{attribute 'GeneratedUsingTerminal: EL2032--0000'}
{attribute addProperty BoxType "EL2032--0000"}
{attribute addProperty Id "DiagAT %I*BOOL1"}
{attribute addProperty CRC "2804620823"}
{attribute addProperty Size "1"}
TYPE Diag_A72B1E17 EXTENDS InputBase_8311D824 :
STRUCT
	{attribute addProperty Name "Diag"}
	Diag AT %I* : BOOL;
END_STRUCT
END_TYPE

(* stored: Version 1.2.0.0, ProductVersion 3.1.4024.9
   DUT Diag_A72B1E17: Id {304d0e0c-4ea6-45d7-93b9-561d30a58be1} *)
